TYPE ST_Identity_PK2_OUT1 :
STRUCT
	ID	:STRING;
	ReadQuality:STRING;
END_STRUCT
END_TYPE

(* stored: Version 1.1.0.1, ProductVersion 3.1.4024.13
   DUT ST_Identity_PK2_OUT1: Id {ab92240e-43c7-46fd-8946-d7847f8e8689} *)
